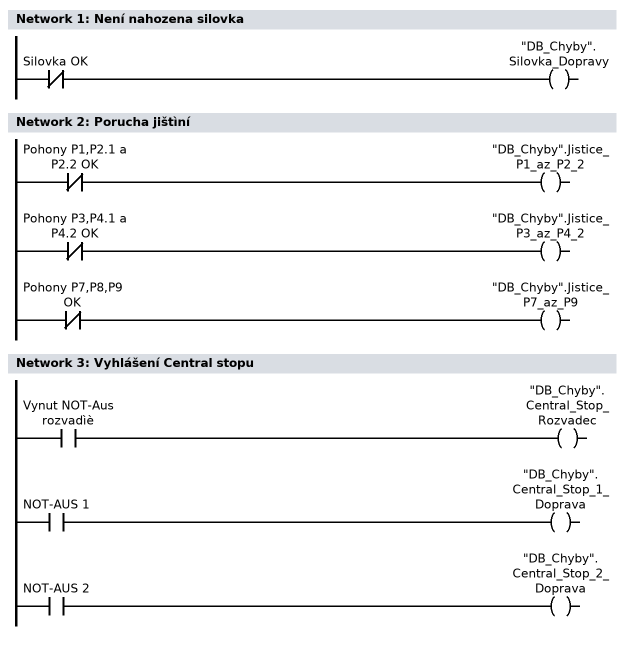
NETWORK
TITLE = Není nahozena silovka 
      AN    "Silovka OK";
      =     "DB_Chyby".Silovka_Dopravy;
NETWORK
TITLE = Porucha jištìní
      AN    "Pohony P1,P2.1 a P2.2 OK";
      =     "DB_Chyby".Jistice_P1_az_P2_2;
      AN    "Pohony P3,P4.1 a P4.2 OK";
      =     "DB_Chyby".Jistice_P3_az_P4_2;
      AN    "Pohony P7,P8,P9 OK";
      =     "DB_Chyby".Jistice_P7_az_P9;
NETWORK
TITLE = Vyhlášení Central stopu
      A     "Vynut NOT-Aus rozvadìè";
      =     "DB_Chyby".Central_Stop_Rozvadec;
      A     "NOT-AUS 1";
      =     "DB_Chyby".Central_Stop_1_Doprava;
      A     "NOT-AUS 2";
      =     "DB_Chyby".Central_Stop_2_Doprava;
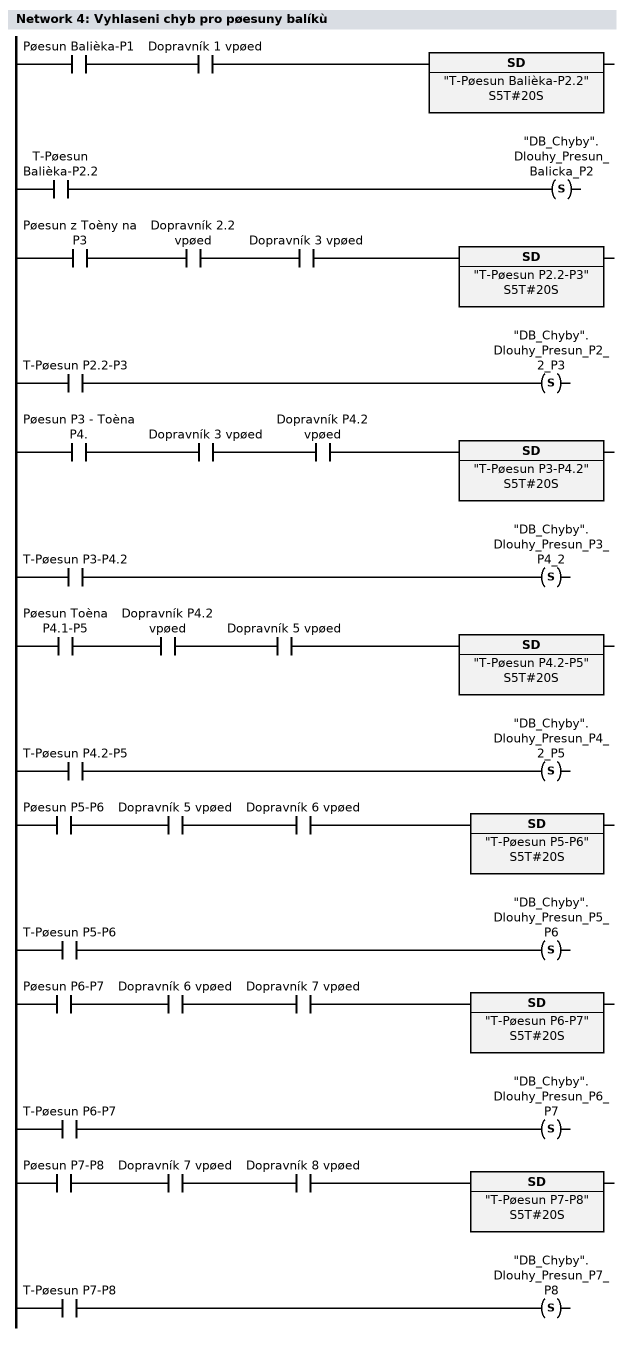
NETWORK
TITLE = Vyhlaseni chyb pro pøesuny balíkù
      A     "Pøesun Balièka-P1";
      A     "Dopravník 1 vpøed";
      L     S5T#20S;
      SD    "T-Pøesun Balièka-P2.2";
      A     "T-Pøesun Balièka-P2.2";
      S     "DB_Chyby".Dlouhy_Presun_Balicka_P2;
      A     "Pøesun z Toèny na P3";
      A     "Dopravník 2.2 vpøed";
      A     "Dopravník 3 vpøed";
      L     S5T#20S;
      SD    "T-Pøesun P2.2-P3";
      A     "T-Pøesun P2.2-P3";
      S     "DB_Chyby".Dlouhy_Presun_P2_2_P3;
      A     "Pøesun P3 - Toèna P4.";
      A     "Dopravník 3 vpøed";
      A     "Dopravník P4.2 vpøed";
      L     S5T#20S;
      SD    "T-Pøesun P3-P4.2";
      A     "T-Pøesun P3-P4.2";
      S     "DB_Chyby".Dlouhy_Presun_P3_P4_2;
      A     "Pøesun Toèna P4.1-P5";
      A     "Dopravník P4.2 vpøed";
      A     "Dopravník 5 vpøed";
      L     S5T#20S;
      SD    "T-Pøesun P4.2-P5";
      A     "T-Pøesun P4.2-P5";
      S     "DB_Chyby".Dlouhy_Presun_P4_2_P5;
      A     "Pøesun P5-P6";
      A     "Dopravník 5 vpøed";
      A     "Dopravník 6 vpøed";
      L     S5T#20S;
      SD    "T-Pøesun P5-P6";
      A     "T-Pøesun P5-P6";
      S     "DB_Chyby".Dlouhy_Presun_P5_P6;
      A     "Pøesun P6-P7";
      A     "Dopravník 6 vpøed";
      A     "Dopravník 7 vpøed";
      L     S5T#20S;
      SD    "T-Pøesun P6-P7";
      A     "T-Pøesun P6-P7";
      S     "DB_Chyby".Dlouhy_Presun_P6_P7;
      A     "Pøesun P7-P8";
      A     "Dopravník 7 vpøed";
      A     "Dopravník 8 vpøed";
      L     S5T#20S;
      SD    "T-Pøesun P7-P8";
      A     "T-Pøesun P7-P8";
      S     "DB_Chyby".Dlouhy_Presun_P7_P8;
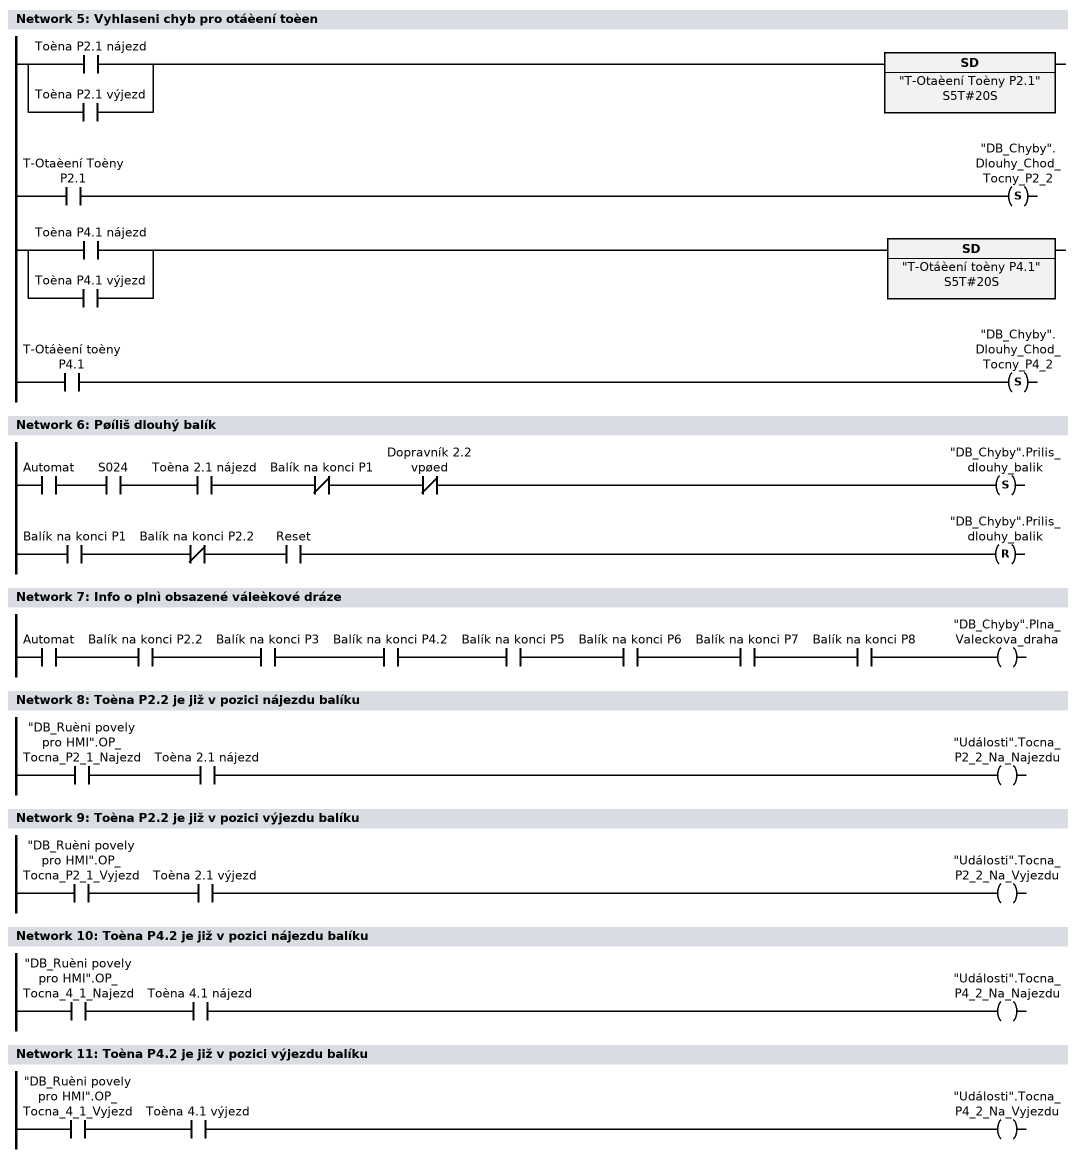
NETWORK
TITLE = Vyhlaseni chyb pro otáèení toèen
      A     "Toèna P2.1 nájezd";
      O;
      A     "Toèna P2.1 výjezd";
      L     S5T#20S;
      SD    "T-Otaèení Toèny P2.1";
      A     "T-Otaèení Toèny P2.1";
      S     "DB_Chyby".Dlouhy_Chod_Tocny_P2_2;
      A     "Toèna P4.1 nájezd";
      O;
      A     "Toèna P4.1 výjezd";
      L     S5T#20S;
      SD    "T-Otáèení toèny P4.1";
      A     "T-Otáèení toèny P4.1";
      S     "DB_Chyby".Dlouhy_Chod_Tocny_P4_2;
NETWORK
TITLE = Pøíliš dlouhý balík
//S010- má obrácenou logiku
      A     "Automat";
      A     "S024";
      A     "Toèna 2.1 nájezd";
      AN    "Balík na konci P1";
      AN    "Dopravník 2.2 vpøed";
      S     "DB_Chyby".Prilis_dlouhy_balik;
      A     "Balík na konci P1";
      AN    "Balík na konci P2.2";
      A     "Reset";
      R     "DB_Chyby".Prilis_dlouhy_balik;
      NOP   0;
NETWORK
TITLE = Info o plnì obsazené váleèkové dráze
      A     "Automat";
      A     "Balík na konci P2.2";
      A     "Balík na konci P3";
      A     "Balík na konci P4.2";
      A     "Balík na konci P5";
      A     "Balík na konci P6";
      A     "Balík na konci P7";
      A     "Balík na konci P8";
      =     "DB_Chyby".Plna_Valeckova_draha;
NETWORK
TITLE = Toèna P2.2 je již v pozici nájezdu balíku
      A     "DB_Ruèni povely pro HMI".OP_Tocna_P2_1_Najezd;
      A     "Toèna 2.1 nájezd";
      =     "Události".Tocna_P2_2_Na_Najezdu;
NETWORK
TITLE = Toèna P2.2 je již v pozici výjezdu balíku
      A     "DB_Ruèni povely pro HMI".OP_Tocna_P2_1_Vyjezd;
      A     "Toèna 2.1 výjezd";
      =     "Události".Tocna_P2_2_Na_Vyjezdu;
NETWORK
TITLE = Toèna P4.2 je již v pozici nájezdu balíku
      A     "DB_Ruèni povely pro HMI".OP_Tocna_4_1_Najezd;
      A     "Toèna 4.1 nájezd";
      =     "Události".Tocna_P4_2_Na_Najezdu;
NETWORK
TITLE = Toèna P4.2 je již v pozici výjezdu balíku
      A     "DB_Ruèni povely pro HMI".OP_Tocna_4_1_Vyjezd;
      A     "Toèna 4.1 výjezd";
      =     "Události".Tocna_P4_2_Na_Vyjezdu;
END_FUNCTION

FUNCTION "Komunikace" : VOID	// FC 50
VERSION : 0.1
BEGIN
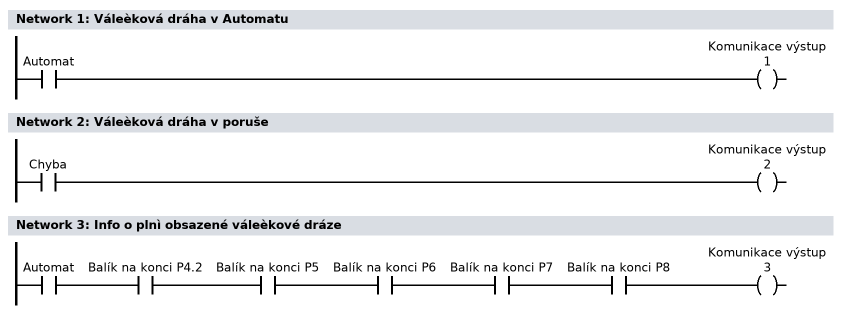
NETWORK
TITLE = Váleèková dráha v Automatu
      A     "Automat";
      =     "Komunikace výstup 1";
NETWORK
TITLE = Váleèková dráha v poruše
      A     "Chyba";
      =     "Komunikace výstup 2";
NETWORK
TITLE = Info o plnì obsazené váleèkové dráze
      A     "Automat";
      A     "Balík na konci P4.2";
      A     "Balík na konci P5";
      A     "Balík na konci P6";
      A     "Balík na konci P7";
      A     "Balík na konci P8";
      =     "Komunikace výstup 3";
END_FUNCTION

DATA_BLOCK "Události"	// DB 100
AUTHOR : Dave
VERSION : 0.1
  STRUCT
   NestandartniOvladani : BOOL ;	//Nestandartni ovladani stroje
   NeniZapnutaSilovka : BOOL ;	//Neni zapnuta silova cast stroje
   Tocna_P2_2_Na_Najezdu : BOOL ;	//Toèna P2.2 je již v pozici nájezdu balíku
   Tocna_P2_2_Na_Vyjezdu : BOOL ;	//Toèna P2.2 je již v pozici výjezdu balíku
   Tocna_P4_2_Na_Najezdu : BOOL ;	//Toèna P4.2 je již v pozici nájezdu balíku
   Tocna_P4_2_Na_Vyjezdu : BOOL ;	//Toèna P4.2 je již v pozici výjezdu balíku
   aaaaa : BOOL ;
   aaaaaa : BOOL ;
   b : BOOL ;
   bb : BOOL ;
   bbb : BOOL ;
   bbbb : BOOL ;
   bbbbb : BOOL ;
   bbbbbb : BOOL ;
   bbbbbbb : BOOL ;
   b7 : BOOL ;
   c : BOOL ;
   c1 : BOOL ;
   c2 : BOOL ;
   c3 : BOOL ;
   c4 : BOOL ;
   c5 : BOOL ;
   c6 : BOOL ;
   c7 : BOOL ;
   d : BOOL ;
   d1 : BOOL ;
   D2 : BOOL ;
   d3 : BOOL ;
   d4 : BOOL ;
   d5 : BOOL ;
   d6 : BOOL ;
   d7 : BOOL ;
   E : DWORD ;
  END_STRUCT ;	
BEGIN
END_DATA_BLOCK

DATA_BLOCK "DB_Chyby"	// DB 101
AUTHOR : Dave
VERSION : 0.1
  STRUCT
   Silovka_Dopravy : BOOL ;	//Nejsou zapnuty silové obvody dopravniku
   Jistice_P1_az_P2_2 : BOOL ;	//Spadený jistiè P1 , P2.1 , P2.2
   Jistice_P3_az_P4_2 : BOOL ;	//Spadený jistiè P3 , P4.1 , P4.2
   Jistice_P7_az_P9 : BOOL ;	//Spadený jistiè P7 , P8 , P9
   Central_Stop_Rozvadec : BOOL ;	//Zmáèknuto Central Stop na rozvadìèi
   Central_Stop_1_Doprava : BOOL ;	//Zmáèknuto Central Stop na dopravnících
   Central_Stop_2_Doprava : BOOL ;	//Zmáèknuto Central Stop na dopravnících
   Dlouhy_Presun_Balicka_P2 : BOOL ;	//Pøíliš dlouhý pøesun balíku z balièky na vstupní dopravník
   Dlouhy_Presun_P2_2_P3 : BOOL ;	//Pøíliš dlouhý pøesun balíku z P2.2 na P3
   Dlouhy_Presun_P3_P4_2 : BOOL ;	//Pøíliš dlouhý pøesun balíku z P3 na P4.2
   Dlouhy_Presun_P4_2_P5 : BOOL ;	//Pøíliš dlouhý pøesun balíku z P4.2 na P5
   Dlouhy_Presun_P5_P6 : BOOL ;	//Pøíliš dlouhý pøesun balíku z P5 na P6
   Dlouhy_Presun_P6_P7 : BOOL ;	//Pøíliš dlouhý pøesun balíku z P6 na P7
   Dlouhy_Presun_P7_P8 : BOOL ;	//Pøíliš dlouhý pøesun balíku z P7 na P8
   Dlouhy_Chod_Tocny_P2_2 : BOOL ;	//Pøíliš dlouhý chod otáèení toèny P2.2
   Dlouhy_Chod_Tocny_P4_2 : BOOL ;	//Pøíliš dlouhý chod otáèení toèny P4.2
   Prilis_dlouhy_balik : BOOL ;	//Pøíliš dlouhý balík
   Plna_Valeckova_draha : BOOL ;	//Valeckova draha je preplnena.
   ccc : BOOL ;
   cccc : BOOL ;
   ccccc : BOOL ;
   cccccc : BOOL ;
   ccccccc : BOOL ;
   cccccccc : BOOL ;
   d : BOOL ;
   dd : BOOL ;
   ddd : BOOL ;
   dddd : BOOL ;
   ddddd : BOOL ;
   dddddd : BOOL ;
   ddddddd : BOOL ;
   dddddddd : BOOL ;
   e : BOOL ;
   ee : BOOL ;
   eee : BOOL ;
   eeee : BOOL ;
   eeeee : BOOL ;
   eeeeee : BOOL ;
   eeeeeee : BOOL ;
   eeeeeeee : BOOL ;
   f : BOOL ;
   ff : BOOL ;
   fff : BOOL ;
   ffff : BOOL ;
   fffff : BOOL ;
   ffffff : BOOL ;
   fffffff : BOOL ;
   ffffffff : BOOL ;
   g : BOOL ;
   gg : BOOL ;
   ggg : BOOL ;
   gggg : BOOL ;
   ggggg : BOOL ;
   gggggg : BOOL ;
   ggggggg : BOOL ;
   gggggggg : BOOL ;
   h : BOOL ;
   hh : BOOL ;
   hhh : BOOL ;
   hhhh : BOOL ;
   hhhhh : BOOL ;
   H5 : BOOL ;
   H6 : BOOL ;
   H7 : BOOL ;
   CH : DWORD ;
   I : DWORD ;
  END_STRUCT ;	
BEGIN
END_DATA_BLOCK

DATA_BLOCK "DB_Ruèni povely pro HMI"	// DB 120
VERSION : 0.1
  STRUCT
   OP_Start_Automatu : BOOL ;	//povel z OP start automatu
   OP_Stop_Automatu : BOOL ;	//povel z OP stop automatu
   OP_Manual : BOOL ;	//povel z OP manualní provoz
   OP_Dopravnik_1_Vpred : BOOL ;	//povel z OP dopravnik vpøed
   OP_Tocna_P2_1_Najezd : BOOL ;	//povel z OP toèna nájezd
   OP_Tocna_P2_1_Vyjezd : BOOL ;	//povel z OP toèna výjezd
   OP_Dopravnik_3_Vpred : BOOL ;	//povel z OP dopravnik vpøed
   OP_Dopravnik_4_Vpred : BOOL ;	//povel z OP dopravnik vpøed
   OP_Tocna_4_1_Najezd : BOOL ;	//povel z OP toèna nájezd
   OP_Tocna_4_1_Vyjezd : BOOL ;	//povel z OP toèna výjezd
   OP_Dopravnik_5_Vpred : BOOL ;	//povel z OP dopravnik vpøed
   OP_Dopravnik_6_Vpred : BOOL ;	//povel z OP dopravnik vpøed
   OP_Dopravnik_7_Vpred : BOOL ;	//povel z OP dopravnik vpøed
   OP_Dopravnik_8_Vpred : BOOL ;	//povel z OP dopravnik vpøed
   bbbbbbb : BOOL ;
   bbbbbbbb : BOOL ;
   c : BOOL ;
   cc : BOOL ;
   ccc : BOOL ;
   cccc : BOOL ;
   ccccc : BOOL ;
   cccccc : BOOL ;
   ccccccc : BOOL ;
   cccccccc : BOOL ;
  END_STRUCT ;	
BEGIN
END_DATA_BLOCK

DATA_BLOCK "DB_Data Hmi"	// DB 140
VERSION : 0.1
  STRUCT
   rez : BOOL ;	//zobrazení chyby stroje
   rez1 : BOOL ;	//zobrazení chyby stroje
   rez2 : BOOL ;	//zobrazení chyby stroje
   rez3 : BOOL ;	//zobrazení chyby stroje
   rez4 : BOOL ;	//zobrazení chyby stroje
   rez5 : BOOL ;	//zobrazení chyby stroje
   rez6 : BOOL ;	//zobrazení chyby stroje
   rez7 : BOOL ;	//zobrazení chyby stroje
   rez8 : BOOL ;	//zobrazení chyby stroje
   rez9 : BOOL ;	//zobrazení chyby stroje
   rez10 : BOOL ;	//zobrazení chyby stroje
   rez12 : BOOL ;	//zobrazení chyby stroje
   rez13 : BOOL ;	//zobrazení chyby stroje
   rezerva1 : BOOL ;
   rezerva2 : BOOL ;
   rezerva3 : BOOL ;
   SystemModeDoprava : INT ;
   SystemStatusRezerva : INT ;
   SystemStatusRezerva_1 : INT ;
  END_STRUCT ;	
BEGIN
END_DATA_BLOCK

ORGANIZATION_BLOCK OB 1
TITLE = "Main Program Sweep (Cycle)"
VERSION : 0.1
VAR_TEMP
  OB1_EV_CLASS : BYTE ;	//Bits 0-3 = 1 (Coming event), Bits 4-7 = 1 (Event class 1)
  OB1_SCAN_1 : BYTE ;	//1 (Cold restart scan 1 of OB 1), 3 (Scan 2-n of OB 1)
  OB1_PRIORITY : BYTE ;	//Priority of OB Execution
  OB1_OB_NUMBR : BYTE ;	//1 (Organization block 1, OB1)
  OB1_RESERVED_1 : BYTE ;	//Reserved for system
  OB1_RESERVED_2 : BYTE ;	//Reserved for system
  OB1_PREV_CYCLE : INT ;	//Cycle time of previous OB1 scan (milliseconds)
  OB1_MIN_CYCLE : INT ;	//Minimum cycle time of OB1 (milliseconds)
  OB1_MAX_CYCLE : INT ;	//Maximum cycle time of OB1 (milliseconds)
  OB1_DATE_TIME : DATE_AND_TIME ;	//Date and time OB1 started
END_VAR
BEGIN
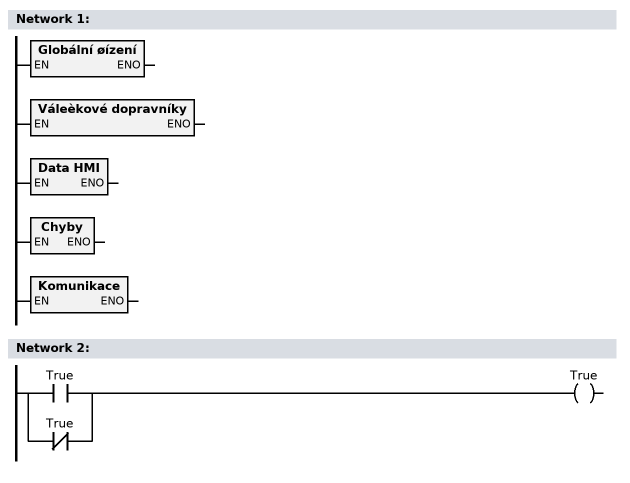
NETWORK
TITLE =
      CALL  "Globální øízení";
      CALL  "Váleèkové dopravníky";
      CALL  "Data HMI";
      CALL  "Chyby";
      CALL  "Komunikace";
NETWORK
TITLE =
      O     "True";
      ON    "True";
      =     "True";
END_ORGANIZATION_BLOCK

ORGANIZATION_BLOCK "CYC_INT5"	// OB 35
TITLE = "Cyclic Interrupt"
VERSION : 0.1
VAR_TEMP
  OB35_EV_CLASS : BYTE ;	//Bits 0-3 = 1 (Coming event), Bits 4-7 = 1 (Event class 1)
  OB35_STRT_INF : BYTE ;	//16#36 (OB 35 has started)
  OB35_PRIORITY : BYTE ;	//Priority of OB Execution
  OB35_OB_NUMBR : BYTE ;	//35 (Organization block 35, OB35)
  OB35_RESERVED_1 : BYTE ;	//Reserved for system
  OB35_RESERVED_2 : BYTE ;	//Reserved for system
  OB35_PHASE_OFFSET : WORD ;	//Phase offset (msec)
  OB35_RESERVED_3 : INT ;	//Reserved for system
  OB35_EXC_FREQ : INT ;	//Frequency of execution (msec)
  OB35_DATE_TIME : DATE_AND_TIME ;	//Date and time OB35 started
END_VAR
BEGIN
// (block stored without names or comments; labels and parameter names are numbered)
END_ORGANIZATION_BLOCK

ORGANIZATION_BLOCK "I/O_FLT1"	// OB 82
TITLE = "I/O Point Fault"
VERSION : 0.1
VAR_TEMP
  OB82_EV_CLASS : BYTE ;	//16#39, Event class 3, Entering event state, Internal fault event
  OB82_FLT_ID : BYTE ;	//16#XX, Fault identifcation code
  OB82_PRIORITY : BYTE ;	//Priority of OB Execution
  OB82_OB_NUMBR : BYTE ;	//82 (Organization block 82, OB82)
  OB82_RESERVED_1 : BYTE ;	//Reserved for system
  OB82_IO_FLAG : BYTE ;	//Input (01010100), Output (01010101)
  OB82_MDL_ADDR : WORD ;	//Base address of module with fault
  OB82_MDL_DEFECT : BOOL ;	//Module defective
  OB82_INT_FAULT : BOOL ;	//Internal fault
  OB82_EXT_FAULT : BOOL ;	//External fault
  OB82_PNT_INFO : BOOL ;	//Point information
  OB82_EXT_VOLTAGE : BOOL ;	//External voltage low
  OB82_FLD_CONNCTR : BOOL ;	//Field wiring connector missing
  OB82_NO_CONFIG : BOOL ;	//Module has no configuration data
  OB82_CONFIG_ERR : BOOL ;	//Module has configuration error
  OB82_MDL_TYPE : BYTE ;	//Type of module
  OB82_SUB_MDL_ERR : BOOL ;	//Sub-Module is missing or has error
  OB82_COMM_FAULT : BOOL ;	//Communication fault
  OB82_MDL_STOP : BOOL ;	//Module is stopped
  OB82_WTCH_DOG_FLT : BOOL ;	//Watch dog timer stopped module
  OB82_INT_PS_FLT : BOOL ;	//Internal power supply fault
  OB82_PRIM_BATT_FLT : BOOL ;	//Primary battery is in fault
  OB82_BCKUP_BATT_FLT : BOOL ;	//Backup battery is in fault
  OB82_RESERVED_2 : BOOL ;	//Reserved for system
  OB82_RACK_FLT : BOOL ;	//Rack fault, only for bus interface module
  OB82_PROC_FLT : BOOL ;	//Processor fault
  OB82_EPROM_FLT : BOOL ;	//EPROM fault
  OB82_RAM_FLT : BOOL ;	//RAM fault
  OB82_ADU_FLT : BOOL ;	//ADU fault
  OB82_FUSE_FLT : BOOL ;	//Fuse fault
  OB82_HW_INTR_FLT : BOOL ;	//Hardware interupt input in fault
  OB82_RESERVED_3 : BOOL ;	//Reserved for system
  OB82_DATE_TIME : DATE_AND_TIME ;	//Date and time OB82 started
END_VAR
BEGIN
// (block stored without names or comments; labels and parameter names are numbered)
END_ORGANIZATION_BLOCK

ORGANIZATION_BLOCK "OBNL_FLT"	// OB 85
TITLE = "Organization Block (OB) Not Loaded Fault"
VERSION : 0.1
VAR_TEMP
  OB85_EV_CLASS : BYTE ;	//16#35 Event class 3
  OB85_FLT_ID : BYTE ;	//16#XX, Fault identification code
  OB85_PRIORITY : BYTE ;	//Priority of OB Execution
  OB85_OB_NUMBR : BYTE ;	//85 (Organization block 85, OB85)
  OB85_RESERVED_1 : BYTE ;	//Reserved for system
  OB85_RESERVED_2 : BYTE ;	//Reserved for system
  OB85_RESERVED_3 : INT ;	//Reserved for system
  OB85_ERR_EV_CLASS : BYTE ;	//Class of event causing error
  OB85_ERR_EV_NUM : BYTE ;	//Number of event causing error
  OB85_OB_PRIOR : BYTE ;	//Priority of OB causing error
  OB85_OB_NUM : BYTE ;	//Number of OB causing error
  OB85_DATE_TIME : DATE_AND_TIME ;	//Date and time OB85 started
END_VAR
BEGIN
// (block stored without names or comments; labels and parameter names are numbered)
END_ORGANIZATION_BLOCK

ORGANIZATION_BLOCK "RACK_FLT"	// OB 86
TITLE = "Loss Of Rack Fault"
VERSION : 0.1
VAR_TEMP
  OB86_EV_CLASS : BYTE ;	//16#38/39 Event class 3
  OB86_FLT_ID : BYTE ;	//16#C1/C4/C5, Fault identifcation code
  OB86_PRIORITY : BYTE ;	//Priority of OB Execution
  OB86_OB_NUMBR : BYTE ;	//86 (Organization block 86, OB86)
  OB86_RESERVED_1 : BYTE ;	//Reserved for system
  OB86_RESERVED_2 : BYTE ;	//Reserved for system
  OB86_MDL_ADDR : WORD ;	//Base address of IM module in rack with fault
  OB86_RACKS_FLTD : ARRAY  [0 .. 31 ] OF BOOL ;	//Racks in fault
  OB86_DATE_TIME : DATE_AND_TIME ;	//Date and time OB86 started
END_VAR
BEGIN
// (block stored without names or comments; labels and parameter names are numbered)
END_ORGANIZATION_BLOCK

ORGANIZATION_BLOCK "Complete Restart"	// OB 100
TITLE = "Complete Restart"
VERSION : 0.1
VAR_TEMP
  OB100_EV_CLASS : BYTE ;	//16#13, Event class 1, Entering event state, Event logged in diagnostic buffer
  OB100_STRTUP : BYTE ;	//16#81/82/83/84 Method of startup
  OB100_PRIORITY : BYTE ;	//Priority of OB Execution
  OB100_OB_NUMBR : BYTE ;	//100 (Organization block 100, OB100)
  OB100_RESERVED_1 : BYTE ;	//Reserved for system
  OB100_RESERVED_2 : BYTE ;	//Reserved for system
  OB100_STOP : WORD ;	//Event that caused CPU to stop (16#4xxx)
  OB100_STRT_INFO : DWORD ;	//Information on how system started
  OB100_DATE_TIME : DATE_AND_TIME ;	//Date and time OB100 started
END_VAR
BEGIN
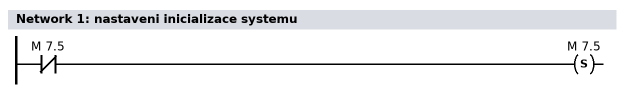
NETWORK
TITLE = nastaveni inicializace systemu
      AN    M 7.5;
      S     M 7.5;
END_ORGANIZATION_BLOCK

ORGANIZATION_BLOCK "Programming Error"	// OB 121
TITLE = "Programming Error"
VERSION : 0.1
VAR_TEMP
  OB121_EV_CLASS : BYTE ;	//16#25, Event class 2, Entering event state, Internal fault event
  OB121_SW_FLT : BYTE ;	//16#XX Software programming fault
  OB121_PRIORITY : BYTE ;	//Priority of OB Execution
  OB121_OB_NUMBR : BYTE ;	//121 (Organization block 121, OB121)
  OB121_BLK_TYPE : BYTE ;	//16#88/8A/8B/8C/8E Type of block fault occured in
  OB121_RESERVED_1 : BYTE ;	//Reserved for system
  OB121_FLT_REG : WORD ;	//16#XX Specific register that caused fault
  OB121_BLK_NUM : WORD ;	//Number of block that programming fault occured in
  OB121_PRG_ADDR : WORD ;	//Address in block where programming fault occured
  OB121_DATE_TIME : DATE_AND_TIME ;	//Date and time OB121 started
END_VAR
BEGIN
// (block stored without names or comments; labels and parameter names are numbered)
END_ORGANIZATION_BLOCK

ORGANIZATION_BLOCK "Module Access Error"	// OB 122
TITLE = "Module Access Error"
VERSION : 0.1
VAR_TEMP
  OB122_EV_CLASS : BYTE ;	//16#29, Event class 2, Entering event state, Internal fault event
  OB122_SW_FLT : BYTE ;	//16#XX Software error code
  OB122_PRIORITY : BYTE ;	//Priority of OB Execution
  OB122_OB_NUMBR : BYTE ;	//122 (Organization block 122, OB122)
  OB122_BLK_TYPE : BYTE ;	//16#88/8C/8E Type of block fault occured in
  OB122_MEM_AREA : BYTE ;	//Memory area where access error occured
  OB122_MEM_ADDR : WORD ;	//Memory address where access error occured
  OB122_BLK_NUM : WORD ;	//Block number in which error occured
  OB122_PRG_ADDR : WORD ;	//Program address where error occured
  OB122_DATE_TIME : DATE_AND_TIME ;	//Date and time OB1 started
END_VAR
BEGIN
// (block stored without names or comments; labels and parameter names are numbered)
END_ORGANIZATION_BLOCK
